{attribute 'OPC.UA.DA' := '1'}
{attribute 'OPC.UA.DA.Access' := '1'}
{attribute 'OPC.UA.DA.StructuredType' := '1'}
TYPE ST_DigitalInput_Sts :
STRUCT
    header   : ST_DeviceHeader_Sts;
    stsValue : BOOL;
END_STRUCT
END_TYPE

(* stored: Version 1.1.0.1, ProductVersion 3.1.4026.12
   DUT ST_DigitalInput_Sts: Id {b0100001-0002-0000-0000-000000000001} *)
